FUNCTION_BLOCK Route IMPLEMENTS iRoute
VAR_INPUT
	
	MotionParameters	: DeltaMotionParameters_typ;	

END_VAR
VAR_OUTPUT
	
	PathBuffer				: ARRAY[0..32767] OF BYTE;
	PathData				: MC_PATH_DATA_REF( ADR( PathBuffer ), SIZEOF( PathBuffer ));

END_VAR
VAR
	
	{attribute 'instance-path'}
	{attribute 'no-init'}
	InstancePath		: STRING;
	
	fbMoveLinearPrep		: MC_MoveLinearAbsolutePreparation;

END_VAR

METHOD AddBlendedPoint : iRoute
VAR_INPUT
	X			: LREAL;
	Y			: LREAL;
	Z			: LREAL;
END_VAR
VAR
	posVector		: ARRAY[0..2] OF LREAL;
	toleranceBall	: ARRAY[0..1] OF LREAL;
END_VAR

// add a single point at the destination
posVector[0]		:= X;
posVector[1]		:= Y;
posVector[2]		:= Z;

// blending radii follows a ratio recommendation from infosys
toleranceBall[0]		:= 0.5 * MotionParameters.BlendingRadius;
toleranceBall[1]		:= MotionParameters.BlendingRadius;

fbMoveLinearPrep.Position			:= ADR( posVector );
fbMoveLinearPrep.PositionCount		:= 3;
fbMoveLinearPrep.Velocity			:= MotionParameters.Velocity;
fbMoveLinearPrep.Acceleration		:= MotionParameters.Acceleration;
fbMoveLinearPrep.Deceleration		:= MotionParameters.Deceleration;
fbMoveLinearPrep.Jerk				:= MotionParameters.Jerk;
fbMoveLinearPrep.BufferMode			:= mcBlendingPrevious;

fbMoveLinearPrep.TransitionMode				:= mcTransModeCornerDistanceAdvanced;
fbMoveLinearPrep.TransitionParameter		:= ADR( toleranceBall );
fbMoveLinearPrep.TransitionParameterCount	:= 2;
fbMoveLinearPrep.InvokeId					:= 100;

fbMoveLinearPrep( PathData := PathData );

// return this for method chaining
AddBlendedPoint		:= THIS^;
END_METHOD

METHOD AddViaPoint : iRoute
VAR_INPUT
	X			: LREAL;
	Y			: LREAL;
	Z			: LREAL;
END_VAR
VAR
	posVector			: ARRAY[0..2] OF LREAL;
END_VAR

// add a single point at the destination
posVector[0]		:= X;
posVector[1]		:= Y;
posVector[2]		:= Z;

fbMoveLinearPrep.Position			:= ADR( posVector );
fbMoveLinearPrep.PositionCount		:= 3;
fbMoveLinearPrep.Velocity			:= MotionParameters.Velocity;
fbMoveLinearPrep.Acceleration		:= MotionParameters.Acceleration;
fbMoveLinearPrep.Deceleration		:= MotionParameters.Deceleration;
fbMoveLinearPrep.Jerk				:= MotionParameters.Jerk;
fbMoveLinearPrep.BufferMode			:= mcBlendingPrevious;

fbMoveLinearPrep.TransitionMode		:= mcTransModeNone;
fbMoveLinearPrep.InvokeId			:= 100;

fbMoveLinearPrep( PathData := PathData );

// return this for method chaining
AddViaPoint		:= THIS^;
END_METHOD

METHOD ClearRoute : iRoute
VAR_INPUT
END_VAR

// clear any existing waypoints in the path buffer
PathData.ClearPath();

// return this for method chaining
ClearRoute		:= THIS^;
END_METHOD

END_FUNCTION_BLOCK

(* stored: Version 1.1.0.1, ProductVersion 3.1.4024.11
   POU Route: Id {713184cf-30c7-46eb-b656-8fb4c47941e5}, SpecialFunc None
   Folder Methods: Id {a0a521d2-cf1d-4900-9367-be85332f3637}
   Folder Properties: Id {8b543435-ae75-47eb-ba22-e51f257b4f70}
   Method AddBlendedPoint: Id {808f2a42-d39a-47ac-95ae-aa8e8bcfee1e}
   Method AddViaPoint: Id {ab1eb623-9748-479b-861d-0ee84722546d}
   Method ClearRoute: Id {994e64ef-ef8a-4802-8672-d451288efe16} *)
